FUNCTION_BLOCK "Station Selection"   // FB20, SCL
{ S7_Optimized_Access := 'TRUE' }
VERSION : 0.1
   VAR_IN_OUT
      settings : "Settings";
      stations : "Stations";
   END_VAR
   VAR
      firstStn : Int;
      rt : "Runtime Data";
      selectionExe : Bool;
      old : Struct
         prevGrp : Bool;
         nextGrp : Bool;
         stnSlct : Array[0..11] of Bool;
      END_STRUCT;
   END_VAR
   VAR_TEMP
      animate : USInt;
      btnPress : Bool;
      count : Int;
      currentBtn : Bool;
      evalObjCount : Int;
      i : Int;
      oldBtn : Bool;
      pStn : Int;
      stnName : WString;
      stnSelected : Bool;
      selState : Bool;
      selStnCount : Int;
      timerExpired : Bool;
      stnSelLblCount : Int;
   END_VAR
   VAR CONSTANT
      ptTimer : Real := 1.5;
   END_VAR
BEGIN
   REGION "UI INTERACTION ANIMATIONS"

       REGION "NEXT GROUP"
           #btnPress := #settings.stations.nextGroup.actuate;
           #animate := "Animate Bool"(colorTrue := "BgLGr",
                                      colorFalse := "BgGray",
                                      evalSignal := #btnPress);
           #settings.stations.nextGroup.animate := #animate;
       END_REGION

       REGION "PREVIOUS GROUP"
           #btnPress := #settings.stations.prevGroup.actuate;
           #animate := "Animate Bool"(colorTrue := "BgLGr",
                                      colorFalse := "BgGray",
                                      evalSignal := #btnPress);
           #settings.stations.prevGroup.animate := #animate;
       END_REGION

       REGION "SELECT ALL STATIONS"
           #btnPress := #settings.stations.selectAll.actuate;
           #animate := "Animate Bool"(colorTrue := "BgLGr",
                                      colorFalse := "BgGray",
                                      evalSignal := #settings.stations.selectAll.actuate);
           #settings.stations.selectAll.animate := #animate;
       END_REGION

   END_REGION

   REGION "POPULATE STATION LABELS"

       REGION "PROCESS NEXT GROUP PRESS"

           REGION "COPY TO LOCAL"
               #currentBtn := #settings.stations.nextGroup.actuate;
               #oldBtn := #old.nextGrp;
           END_REGION

           REGION "FALLING EDGE OF NEXT GROUP"
               IF NOT #currentBtn AND #oldBtn THEN

                   REGION "INCREMENT FIRST STATION"
                       #firstStn := #firstStn + 2;
                   END_REGION

                   REGION "UPPER LIMIT ROLL OVER"
                       IF #firstStn > "stnCount" THEN
                           #firstStn := #firstStn - "stnCount" - 1;
                       END_IF;
                   END_REGION

               END_IF;
           END_REGION

           REGION "NEXT GROUP CHANGE DETECTION"
               #old.nextGrp := #currentBtn;
           END_REGION

       END_REGION

       REGION "PROCESS PREVIOUS GROUP PRESS"

           REGION "COPY TO LOCAL"
               #currentBtn := #settings.stations.prevGroup.actuate;
               #oldBtn := #old.prevGrp;
           END_REGION

           REGION "FALLING EDGE OF PREVIOUS GROUP"
               IF NOT #currentBtn AND #oldBtn THEN

                   REGION "DECREMENT FIRST STATION"
                       #firstStn := #firstStn - 2;
                   END_REGION

                   REGION "LOWER LIMIT ROLL OVER"
                       IF #firstStn < 0 THEN
                           #firstStn := #firstStn + "stnCount" + 1;
                       END_IF;
                   END_REGION

               END_IF;
           END_REGION

           REGION "PREVIOUS GROUP CHANGE DETECTION"
               #old.prevGrp := #currentBtn;
           END_REGION

       END_REGION

       REGION "WRITE LABEL"

           REGION "COPY TO LOCAL"
               #evalObjCount := "hmiSelStnCount";
           END_REGION

           REGION "FOR EACH STATION SELECTION BUTTON"
               FOR #i := 0 TO #evalObjCount DO

                   REGION "CALCULATE POINTER"
                       #pStn := #firstStn + #i;
                   END_REGION

                   REGION "UPPER LIMIT ROLL OVER"
                       IF #pStn > "stnCount" THEN
                           #pStn := #firstStn + #i - "stnCount" - 1;
                       END_IF;
                   END_REGION

                   REGION "BUILD NAME"
                       #stnName := CONCAT_WSTRING(IN1 := #stations.me[#pStn].line,
                                                  IN2 := wstring#' ',
                                                  IN3 := "Strip Sign"(USINT_TO_WSTRING(#stations.me[#pStn].dropZone)));
                   END_REGION

                   REGION "WRITE NAME"
                       #settings.stations.selectBtns[#i].label := #stnName;
                   END_REGION

               END_FOR;
           END_REGION

       END_REGION

   END_REGION

   REGION "SINGLE STATION SELECTION"

       REGION "COPY TO LOCAL"
           #stnSelLblCount := "hmiSelStnCount";
       END_REGION

       REGION "LOOP THROUGH DISPLAYED STATIONS"
           FOR #i := 0 TO #stnSelLblCount DO

               REGION "CALCULATE POINTER"
                   #pStn := #firstStn + #i;
               END_REGION

               REGION "UPPER LIMIT ROLL OVER"
                   IF #pStn > "stnCount" THEN
                       #pStn := #firstStn + #i - "stnCount" - 1;
                   END_IF;
               END_REGION

               REGION "COPY TO LOCAL"
                   #currentBtn := #settings.stations.selectBtns[#i].actuate;
                   #oldBtn := #old.stnSlct[#i];
               END_REGION

               REGION "TOGGLE STATE ON FALLING EDGE"
                   IF NOT #currentBtn AND #oldBtn THEN
                       #selState := #stations.me[#pStn].settings.selected;
                       #selState := NOT #selState;
                       #stations.me[#pStn].settings.selected := #selState;
                   END_IF;
               END_REGION

               REGION "STATION SELECTION CHANGE DETECTION"
                   #old.stnSlct[#i] := #currentBtn;
               END_REGION

           END_FOR;
       END_REGION

   END_REGION

   REGION "MULTI SELECT TIMER"

       REGION "RUNTIME CALL"
           #rt.elapsed := RUNTIME(#rt.mem);
       END_REGION

       REGION "TIMER"

           REGION "COPY TO LOCAL"
               #btnPress := #settings.stations.selectAll.actuate;
           END_REGION

           REGION "ACCUMULATE RT VALUES"
               IF #btnPress THEN
                   #rt.asReal += LREAL_TO_REAL(#rt.elapsed);
               END_IF;
           END_REGION

           REGION "SET TIMER FLAG"
               IF #rt.asReal < #ptTimer THEN
                   #timerExpired := FALSE;
               END_IF;
               IF #rt.asReal >= #ptTimer THEN
                   #timerExpired := TRUE;
                   #rt.asReal := 0.0;
               END_IF;
           END_REGION

           REGION "RESET ACCUMULATED VALUE"
               IF NOT #btnPress THEN
                   #rt.asReal := 0.0;
                   #selectionExe := FALSE;
               END_IF;
           END_REGION

       END_REGION

   END_REGION

   REGION "EVALUATE MULTI SELECTION"
       IF #timerExpired AND NOT #selectionExe THEN

           REGION "COPY TO LOCAL"
               #selStnCount := #settings.stations.selCount;
           END_REGION

           REGION "SELECT ALL"
               IF #selStnCount < "stnCount" THEN
                   "Select Stations"(mode := TRUE,
                                     stations := #stations);
               END_IF;
           END_REGION

           REGION "DESELECT ALL"
               IF #selStnCount = "stnCount" THEN
                   "Select Stations"(mode := FALSE,
                                     stations := #stations);
               END_IF;
           END_REGION

           REGION "FLAG SELECTION EXECUTED"
               #selectionExe := TRUE;
           END_REGION

       END_IF;
   END_REGION

   REGION "SELECTION ANIMATIONS"

       REGION "COPY TO LOCAL"
           #stnSelLblCount := "hmiSelStnCount";
       END_REGION

       REGION "LOOP THROUGH BUTTONS"
           FOR #i := 0 TO #stnSelLblCount DO

               REGION "CALCULATE POINTER"
                   #pStn := #firstStn + #i;
               END_REGION

               REGION "UPPER LIMIT ROLL OVER"
                   IF #pStn > "stnCount" THEN
                       #pStn := #firstStn + #i - "stnCount" - 1;
                   END_IF;
               END_REGION

               REGION "COPY TO LOCAL"
                   #currentBtn := #settings.stations.selectBtns[#i].actuate;
                   #stnSelected := #stations.me[#pStn].settings.selected;
               END_REGION

               REGION "DRAW SELCTION HIGHLIGHTS"
                   #animate := "Animate Bool"(colorTrue := "BgLTe",
                                              colorFalse := "BgGray",
                                              evalSignal := #stnSelected);
               END_REGION

               REGION "ANIMATE BUTTON PRESS"
                   #animate := "Animate Bool"(colorTrue := "BgDTe",
                                              colorFalse := #animate,
                                              evalSignal := #currentBtn);
                   #settings.stations.selectBtns[#i].animate := #animate;
               END_REGION

           END_FOR;
       END_REGION

   END_REGION

   REGION "COUNT SELECTED STATIONS"

       REGION "INITIALIZE LOCAL"
           #count := 0;
           #evalObjCount := "stnCount";
       END_REGION

       REGION "LOOP THROUGH STATIONS"
           FOR #i := 0 TO #evalObjCount DO

               REGION "INCREMENT COUNT ON SELECTION"
                   #stnSelected := #stations.me[#i].settings.selected;
                   IF #stnSelected THEN
                       #count += 1;
                   END_IF;
               END_REGION

           END_FOR;
       END_REGION

       REGION "SAVE COUNT"
           #settings.stations.selCount := #count;
       END_REGION

   END_REGION
END_FUNCTION_BLOCK

FUNCTION_BLOCK "KP8 Button Selections"   // FB21, SCL
{ S7_Optimized_Access := 'TRUE' }
VERSION : 0.1
   VAR_INPUT
      reset : Bool;
   END_VAR
   VAR_IN_OUT
      settings : "Settings";
      stations : "Stations";
   END_VAR
   VAR
      enableState : Bool;
      oldBtnPresses : Array[0..7] of Bool;
      oldSelState : Array[0..7] of Bool;
      oldSelStnCount : Int;
      rt : "Runtime Data";
      timerExpired : Bool;
      selectionExe : Bool;
   END_VAR
   VAR_TEMP
      animate : USInt;
      btnPress : Bool;
      count : Int;
      i : Int;
      j : Int;
      mode : Bool;
      oldPress : Bool;
      pBtn : Int;
      selBtnCount : Int;
      selStnCount : Int;
      stnSelected : Bool;
   END_VAR
   VAR CONSTANT
      selectAllTime : Real := 1.5;
   END_VAR
BEGIN
   REGION "ENABLE KP8 BUTTON ASSIGNMENT SECTION"

       REGION "ENABLE"

           REGION "COPY TO LOCAL"
               #selStnCount := #settings.stations.selCount;
           END_REGION

           REGION "ON CHANGE IN SELECTED STATION COUNT"
               IF #selStnCount <> 0 AND #selStnCount <> #oldSelStnCount THEN

                   REGION "ENABLE KP8 SELECTIONS"
                       #enableState := TRUE;
                   END_REGION

               END_IF;
           END_REGION

       END_REGION

       REGION "DISABLE"

           REGION "COPY TO LOCAL"
               #selStnCount := #settings.stations.selCount;
           END_REGION

           REGION "ON DESELETION OF LAST STATION"
               IF #selStnCount = 0 AND #selStnCount <> #oldSelStnCount THEN

                   REGION "RESET ENABLED STATE"
                       #enableState := FALSE;
                   END_REGION

                   REGION "RESET BUTTON SELECTION STATES"
                       FOR #i := 0 TO "ptsPerStn" DO
                           #settings.kp8.btnSelState[#i] := FALSE;
                       END_FOR;
                   END_REGION

               END_IF;
           END_REGION

       END_REGION

   END_REGION

   REGION "SINGLE BUTTON SELECTION"

       REGION "LOOP THROUGH BUTTONS"
           FOR #i := 0 TO "ptsPerStn" DO

               REGION "EXCLUDE STOP RUNTIME AND RESET SELECTED BUTTONS"
                   IF #i <> 0 AND #i <> 4 THEN

                       REGION "COPY TO LOCAL"

                           REGION "CALCULATE BUTTON POINTER"
                               CASE #i OF
                                   1:
                                       #pBtn := 5;
                                   2:
                                       #pBtn := 3;
                                   3:
                                       #pBtn := 1;
                                   5:
                                       #pBtn := 4;
                                   6:
                                       #pBtn := 2;
                                   7:
                                       #pBtn := 0;
                                   ELSE
                                       ;
                               END_CASE;
                           END_REGION

                           #btnPress := #settings.kp8.buttons[#i].actuate OR #settings.viewingStation.btns[#pBtn].select.actuate;
                           #oldPress := #oldBtnPresses[#i];

                       END_REGION

                       REGION "TOGGLE STATE ON FALLING EDGE"
                           IF NOT #btnPress AND #oldPress THEN
                               #settings.kp8.btnSelState[#i] := NOT #settings.kp8.btnSelState[#i];
                               #settings.kp8.selBtnNumber := #i;
                           END_IF;
                       END_REGION

                       REGION "SAVE SELECTED BUTTON NUMBER ON DESELECT"
                           IF NOT #settings.kp8.btnSelState[#i] AND #oldSelState[#i] THEN
                               FOR #j := 0 TO "ptsPerStn" DO
                                   IF #settings.kp8.btnSelState[#j] THEN
                                       #settings.kp8.selBtnNumber := #j;
                                   END_IF;
                               END_FOR;
                           END_IF;
                       END_REGION

                       REGION "KP8 BUTON SELECTION CHANGE DETECTION"
                           #oldBtnPresses[#i] := #btnPress;
                       END_REGION

                   END_IF;
               END_REGION

           END_FOR;
       END_REGION

   END_REGION

   REGION "MULTI BUTTON SELECTION"

       REGION "MULTI SELECT TIMER"

           REGION "RUNTIME CALL"
               #rt.elapsed := RUNTIME(#rt.mem);
           END_REGION

           REGION "TIMER"

               REGION "COPY TO LOCAL"
                   #btnPress := #settings.kp8.selectButtons.actuate;
               END_REGION

               REGION "ACCUMULATE RT VALUES"
                   IF #btnPress THEN
                       #rt.asReal += LREAL_TO_REAL(#rt.elapsed);
                   END_IF;
               END_REGION

               REGION "SET TIMER FLAG"
                   IF #rt.asReal < #selectAllTime THEN
                       #timerExpired := FALSE;
                   END_IF;
                   IF #rt.asReal >= #selectAllTime THEN
                       #timerExpired := TRUE;
                       #rt.asReal := 0.0;
                   END_IF;
               END_REGION

               REGION "RESET ACCUMULATED VALUE"
                   IF NOT #btnPress THEN
                       #rt.asReal := 0.0;
                       #selectionExe := FALSE;
                   END_IF;
               END_REGION

           END_REGION

       END_REGION

       REGION "EVALUATE MULTI SELECTION"
           IF #timerExpired AND NOT #selectionExe THEN

               REGION "COPY TO LOCAL"
                   #selBtnCount := #settings.kp8.selCount;
               END_REGION

               REGION "SELECT ALL"
                   IF #selBtnCount < "ptsPerStn" - 1 THEN
                       #mode := TRUE;
                   END_IF;
               END_REGION

               REGION "DESELECT ALL"
                   IF #selBtnCount = "ptsPerStn" - 1 THEN
                       #mode := FALSE;
                   END_IF;
               END_REGION

               REGION "SAVE SELECTIONS"
                   FOR #i := 0 TO "ptsPerStn" DO

                       REGION "EXCLUDE STOP RUNTIME AND RESET SELECTED BUTTONS"
                           IF #i <> 0 AND #i <> 4 THEN

                               REGION "PERFROM SELECTION"
                                   #settings.kp8.btnSelState[#i] := #mode;
                               END_REGION

                           END_IF;
                       END_REGION

                   END_FOR;
               END_REGION

               REGION "SET SELECED BUTTON NUMBER TO 1"
                   #settings.kp8.selBtnNumber := 0;
               END_REGION

               REGION "FLAG SELECTION EXECUTED"
                   #selectionExe := TRUE;
               END_REGION

           END_IF;
       END_REGION
   END_REGION

   REGION "SAVE BUTTON SELECTIONS TO STATIONS"

       REGION "COPY TO LOCAL"
           #selStnCount := #settings.stations.selCount;
       END_REGION

       REGION "ON CHANGE IN BUTTON OR STATION SELECTON"
           IF #settings.kp8.btnSelState <> #oldSelState OR #selStnCount <> #oldSelStnCount THEN

               REGION "FOR SELECTED STATIONS"
                   FOR #i := 0 TO "stnCount" DO
                       #stnSelected := #stations.me[#i].settings.selected;
                       IF #stnSelected THEN

                           REGION "SAVE BUTTON SELECTION STATE"
                               #stations.me[#i].settings.btnSelection := #settings.kp8.btnSelState;
                           END_REGION

                       END_IF;
                   END_FOR;
               END_REGION

           END_IF;
       END_REGION

       REGION "SELECTED STATION COUNT CHANGE DETECTION"
           #oldSelStnCount := #selStnCount; 
       END_REGION

   END_REGION

   REGION "COUNT SELECTED BUTTONS"

       REGION "ON CHANGE IN BUTTON SELECTION STATES"
           IF #settings.kp8.btnSelState <> #oldSelState THEN

               REGION "INITIALIZE LOCAL"
                   #count := 0;
               END_REGION

               REGION "FOR EACH SELECTED BUTTON"
                   FOR #i := 0 TO "ptsPerStn" DO
                       IF #settings.kp8.btnSelState[#i] THEN

                           REGION "INCREMENT COUNT"
                               #count := #count + 1;
                           END_REGION

                       END_IF;
                   END_FOR;
               END_REGION

               REGION "SAVE COUNT"
                   #settings.kp8.selCount := #count;
               END_REGION

           END_IF;
       END_REGION

   END_REGION 

   REGION "UI INTERACTION ANIMATIONS"

       REGION "SELECT ALL BUTTONS"
           #btnPress := #settings.kp8.selectButtons.actuate;
           #animate := "Animate Bool"(colorTrue := "BgLGr",
                                      colorFalse := "BgGray",
                                      evalSignal := #btnPress);
           #settings.kp8.selectButtons.animate := #animate;
       END_REGION

       REGION "STOP RESET SELECTED STATION"
           #btnPress := #settings.kp8.buttons[0].actuate;
           #animate := "Animate Bool"(colorTrue := "FgGray",
                                      colorFalse := "BgGray",
                                      evalSignal := #btnPress);
           #settings.kp8.buttons[0].animate := #animate;
       END_REGION

       REGION "STOP RUNTIME"
           #btnPress := #settings.kp8.buttons[4].actuate;
           #animate := "Animate Bool"(colorTrue := "FgGray",
                                      colorFalse := "BgGray",
                                      evalSignal := #btnPress);
           #settings.kp8.buttons[4].animate := #animate;
       END_REGION

       REGION "BUTTON SELECTIONS"

           REGION "FOR EACH BUTTON"     
               FOR #i := 0 TO "ptsPerStn" DO

                   REGION "EXCLUDE STOP RUNTIME AND RESET SELECTED BUTTONS"
                       IF #i <> 0 AND #i <> 4 THEN

                           REGION "ANIMATE"

                               REGION "COPY TO LOCAL"
                                   #btnPress := #settings.kp8.buttons[#i].actuate;
                               END_REGION

                               REGION "ENABLE/DISABLE"
                                   #animate := "Animate Bool"(colorTrue := "BgGray",
                                                              colorFalse := "disabled",
                                                              evalSignal := #enableState);
                               END_REGION

                               REGION "ENABLED SUB ANIMATIONS"
                                   IF #enableState THEN

                                       REGION "BUTTON SELECTED"
                                           #animate := "Animate Bool"(colorTrue := "BgLTe",
                                                                      colorFalse := #animate,
                                                                      evalSignal := #settings.kp8.btnSelState[#i]);
                                       END_REGION

                                       REGION "BUTTON UP/DOWN"
                                           #animate := "Animate Bool"(colorTrue := "BgDTe",
                                                                      colorFalse := #animate,
                                                                      evalSignal := #btnPress);
                                       END_REGION
                                   END_IF;
                               END_REGION

                               REGION "SAVE ANIMATION"
                                   #settings.kp8.buttons[#i].animate := #animate;
                               END_REGION

                           END_REGION

                       END_IF;
                   END_REGION

               END_FOR;
           END_REGION

       END_REGION

   END_REGION

   REGION "DRAW KP8 BUTTON LABELS"
       IF #reset THEN
           #settings.kp8.buttons[1].label := wstring#'6';
           #settings.kp8.buttons[2].label := wstring#'4';
           #settings.kp8.buttons[3].label := wstring#'2';
           #settings.kp8.buttons[5].label := wstring#'5';
           #settings.kp8.buttons[6].label := wstring#'3';
           #settings.kp8.buttons[7].label := wstring#'1';
       END_IF;
   END_REGION

   REGION "CHANGE DETECTION"
       #oldSelState := #settings.kp8.btnSelState;
   END_REGION
END_FUNCTION_BLOCK

FUNCTION_BLOCK "Buffer Log: Part Requests"   // FB22, SCL
{ S7_Optimized_Access := 'TRUE' }
VERSION : 0.1
   VAR_INPUT
      stations : "Stations";
   END_VAR
   VAR_IN_OUT
      logBuffer : "Part Req Log";
      logFlag : Int;
   END_VAR
   VAR
      clpsLogTime : Real;
      old : Struct
         ordered : "Station Old Presses";
         requested : "Station Old Presses";
      END_STRUCT;
      pLogBuffer : Int;
      rt : "Runtime Data";
   END_VAR
   VAR_TEMP
      address : Int;
      btnCount : Int;
      clpsFlag : Bool;
      i : Int;
      j : Int;
      oldPartOrdered : Bool;
      oldPartReq : Bool;
      partOrdered : Bool;
      partReq : Bool;
      stnCount : Int;
      readTimeRetVal : Int;
      blankRow : "Part Req Log Row";
   END_VAR
   VAR CONSTANT
      clpsItrvl : Real := 2.0;
      fulfilled : Int := 3;
      ordered : Int := 2;
      requested : Int := 1;
   END_VAR
BEGIN
   REGION "RUNTIME CALL"
       #rt.elapsed := RUNTIME(#rt.mem);
       #rt.asReal := LREAL_TO_REAL(#rt.elapsed);
   END_REGION

   REGION "COPY TO LOCAL"
       #btnCount := "ptsPerStn";
       #stnCount := "stnCount";
   END_REGION

   REGION "FOR EACH STATION"
       FOR #i := 0 TO #stnCount DO

           REGION "FOR EACH BUTTON"
               FOR #j := 0 TO #btnCount DO

                   REGION "COPY TO LOCAL"
                       #partOrdered := #stations.me[#i].partOrdered[#j];
                       #partReq := #stations.me[#i].partRequested[#j];
                       #oldPartOrdered := #old.ordered.me[#i,#j];
                       #oldPartReq := #old.requested.me[#i,#j];
                   END_REGION;

                   REGION "CALCULATE ADDRESS"
                       #address := (#i + 1) * 10 + #j + 1;
                   END_REGION

                   REGION "ON PART REQUEST RISING EDGE"
                       IF #partReq AND NOT #oldPartReq THEN

                           REGION "LOG ENTRY"
                               #logBuffer.me[#pLogBuffer] := "Buffer Part Req Log Row: Generate"(address := #address,
                                                                                        type := #requested);
                           END_REGION

                           REGION "INCREMENT POINTER"
                               #pLogBuffer += 1;
                           END_REGION

                       END_IF;
                   END_REGION

                   REGION "ON PART ORDERED RISING EDGE"
                       IF #partOrdered AND NOT #oldPartOrdered THEN

                           REGION "REQUEST TYPE"
                               #logBuffer.me[#pLogBuffer] := "Buffer Part Req Log Row: Generate"(address := #address,
                                                                                                 type := #ordered);
                           END_REGION

                           REGION "INCREMENT POINTER"
                               #pLogBuffer += 1;
                           END_REGION

                       END_IF;
                   END_REGION

                   REGION "ON PART REQUEST FALLING EDGE"
                       IF NOT #partReq AND #oldPartReq THEN

                           REGION "REQUEST TYPE"
                               #logBuffer.me[#pLogBuffer] := "Buffer Part Req Log Row: Generate"(
                                   address := #address,
                                   type := #fulfilled
                               );
                           END_REGION

                           REGION "INCREMENT POINTER"
                               #pLogBuffer += 1;
                           END_REGION

                       END_IF;
                   END_REGION

                   REGION "SAVE FOR CHANGE DETECTION"
                       #old.requested.me[#i, #j] := #partReq;
                       #old.ordered.me[#i, #j] := #partOrdered;
                   END_REGION

               END_FOR;
           END_REGION

       END_FOR;
   END_REGION

   REGION "SEND TO HMI"

       REGION "ON ENTRY IN BUFFER"
           IF #logBuffer.me[0].address <> 0 THEN

               REGION "TIMER"
                   #clpsLogTime += #rt.asReal;
                   IF #clpsLogTime >= #clpsItrvl THEN
                       #clpsLogTime := 0.0;
                       #clpsFlag := TRUE;
                   END_IF;
               END_REGION

               REGION "EXECUTE COLLAPSE"
                   IF #clpsFlag THEN

                       REGION "MOVE BUFFER UP ONE POSITION"
                           FOR #i := 0 TO 98 DO
                               #logBuffer.me[#i] := #logBuffer.me[#i + 1];
                           END_FOR;
                       END_REGION

                       REGION "DELETE LAST ROW"
                           #logBuffer.me[99] := #blankRow;
                       END_REGION

                       REGION "FLAG FOR HMI"
                           #logFlag += 1;
                           IF #logFlag > 9 THEN
                               #logFlag := 0;
                           END_IF;
                       END_REGION

                       REGION "DECREMENT POINTER"
                           #pLogBuffer -= 1;
                       END_REGION

                   END_IF;
               END_REGION

           END_IF;
       END_REGION

   END_REGION

   REGION "RESET TIMER"
       IF #logBuffer.me[0].address = 0 THEN
           #clpsLogTime := 0.0;
       END_IF;
   END_REGION
END_FUNCTION_BLOCK

FUNCTION_BLOCK "Enable Assignment Pair"   // FB23, SCL
{ S7_Optimized_Access := 'TRUE' }
VERSION : 0.1
   VAR_INPUT
      disable : Bool;
      enable : Bool;
   END_VAR
   VAR_IN_OUT
      value : WString;
      assignAnimate : USInt;
      ioFieldAnimate : USInt;
   END_VAR
   VAR
      old : Struct
         disabled : Bool;
         enabled : Bool;
      END_STRUCT;
   END_VAR
BEGIN
   REGION "DISABLED"    
       IF #disable THEN
           #value := wstring#'';
           #assignAnimate := "disabled";
           #ioFieldAnimate := "disabled";
       END_IF;
   END_REGION

   REGION "ENABLED"
           IF #enable THEN
               #assignAnimate := "BgGray";
               #ioFieldAnimate := "BgWh";
           END_IF;
   END_REGION
END_FUNCTION_BLOCK

FUNCTION_BLOCK "Assign Button Parameters"   // FB24, SCL
{ S7_Optimized_Access := 'TRUE' }
VERSION : 0.1
   VAR_INPUT
      settings : "Settings";
   END_VAR
   VAR_IN_OUT
      stations : "Stations";
   END_VAR
   VAR
      old : Struct
         allotted : Bool;
         critical : Bool;
         pn : Bool;
      END_STRUCT;
   END_VAR
   VAR_TEMP
      assign : Bool;
      btn : Struct
         allotted : Bool;
         critical : Bool;
         pn : Bool;
      END_STRUCT;
      btnSelected : Bool;
      i : Int;
      j : Int;
      partNumber : WString;
      stnSelected : Bool;
      timerReal : Real;
   END_VAR
BEGIN
   REGION "COPY TO LOCACL"
       #btn.allotted := #settings.alotted.assign.actuate;
       #btn.critical := #settings.critical.assign.actuate;
       #btn.pn := #settings.partNumber.assign.actuate;
   END_REGION

   REGION "ASSIGNMENT PULSE"
       #assign := (#btn.allotted AND NOT #old.allotted)
                   OR (#btn.critical AND NOT #old.critical)
                   OR (#btn.pn AND NOT #old.pn);
   END_REGION

   REGION "ON ASSIGNMENT PULSE"
       IF #assign THEN
           REGION "PROCESS VARIABLE"

               REGION "PART NUMBER"
                   IF #btn.pn THEN
                       #partNumber := #settings.partNumber.ioField.value;
                   END_IF;
               END_REGION

               REGION "CRITICAL TIME"
                   IF #btn.critical THEN
                       #timerReal := "WString Timer to Real"(#settings.critical.ioField.value);
                   END_IF;
               END_REGION

               REGION "ALLOTTED TIME"
                   IF #btn.allotted THEN
                       #timerReal := "WString Timer to Real"(#settings.alotted.ioField.value);
                   END_IF;
               END_REGION

           END_REGION

           REGION "FOR EACH STATION"
               FOR #i := 0 TO "stnCount" DO

                   REGION "COPY TO LOCAL"
                       #stnSelected := #stations.me[#i].settings.selected;
                   END_REGION

                   REGION "ON SELECTED STATION"
                       IF #stnSelected THEN

                           REGION "FOR EACH BUTTON"
                               FOR #j := 0 TO "ptsPerStn" DO

                                   REGION "COPY TO LOCAL"
                                       #btnSelected := #stations.me[#i].settings.btnSelection[#j];
                                   END_REGION

                                   REGION "ON SELECTED BUTTON"
                                       IF #btnSelected THEN

                                           REGION "ASSIGN PART NUMBER"
                                               IF #btn.pn THEN
                                                   #stations.me[#i].partNumbers[#j] := #partNumber;
                                               END_IF;
                                           END_REGION

                                           REGION "ASSIGN ALLOTTED TIME"
                                               IF #btn.allotted THEN
                                                   #stations.me[#i].presetTime.allotted[#j] := #timerReal;
                                               END_IF;
                                           END_REGION

                                           REGION "ASSIGN CRITICAL TIME"
                                               IF #btn.critical THEN
                                                   #stations.me[#i].presetTime.critical[#j] := #timerReal;
                                               END_IF;
                                           END_REGION

                                       END_IF;
                                   END_REGION

                               END_FOR;
                           END_REGION

                       END_IF;
                   END_REGION

               END_FOR;
           END_REGION

       END_IF;
   END_REGION

   REGION "CHANGE DETECTION"
       #old := #btn;
   END_REGION
END_FUNCTION_BLOCK

FUNCTION_BLOCK "Animate: PN & Timers"   // FB25, SCL
{ S7_Optimized_Access := 'TRUE' }
VERSION : 0.1
   VAR_INPUT
      stations : "Stations";
   END_VAR
   VAR_IN_OUT
      settings : "Settings";
   END_VAR
   VAR
      instPNEntEnable : "Enable Assignment Pair";
      instAlltEntEnable : "Enable Assignment Pair";
      instCrtEntEnable : "Enable Assignment Pair";
   END_VAR
   VAR_TEMP
      animate : USInt;
      disable : Bool;
      enable : Bool;
      selBtnCount : Int;
      selStnCount : Int;
   END_VAR
BEGIN
   REGION "COPY TO LOCAL"
       #selBtnCount := #settings.kp8.selCount;
       #selStnCount := #settings.stations.selCount;
   END_REGION

   REGION "ENABLE/DISABLE FOR PN AND TIMERS"

       REGION "SET DISABLE"
           IF #selStnCount = 0 OR #selBtnCount = 0 THEN
               #disable := TRUE;
               #enable := FALSE;
           END_IF;
       END_REGION

       REGION "SET ENABLE"
           IF #selStnCount <> 0 AND #selBtnCount <> 0 THEN
               #disable := FALSE;
               #enable := TRUE;
           END_IF;
       END_REGION

   END_REGION

   REGION "PN ANIMATION FUNCTIONS"
       #animate := #settings.partNumber.assign.animate;
       #instPNEntEnable(disable := #disable,
                        enable := #enable,
                        value := #settings.partNumber.ioField.value,
                        assignAnimate := #animate,
                        ioFieldAnimate := #settings.partNumber.ioField.animate);
       #animate := "Animate Bool"(colorTrue := "BgLGr",
                                  colorFalse := #animate,
                                  evalSignal := #settings.partNumber.assign.actuate);
       #settings.partNumber.assign.animate := #animate;
   END_REGION

   REGION "ALLOTTED TIME ANIMATION FUNCTIONS"
       #animate := #settings.alotted.assign.animate;
       #instAlltEntEnable(disable := #disable,
                          enable := #enable,
                          value := #settings.alotted.ioField.value,
                          assignAnimate := #animate,
                          ioFieldAnimate := #settings.alotted.ioField.animate);
       #animate := "Animate Bool"(colorTrue := "BgLGr",
                                  colorFalse := #animate,
                                  evalSignal := #settings.alotted.assign.actuate);
       #settings.alotted.assign.animate := #animate;
   END_REGION

   REGION "CRITICAL TIME ANIMATION FUNCTIONS"
       #animate := #settings.critical.assign.animate;
       #instCrtEntEnable(disable := #disable,
                         enable := #enable,
                         value := #settings.critical.ioField.value,
                         assignAnimate := #animate,
                         ioFieldAnimate := #settings.critical.ioField.animate);
       #animate := "Animate Bool"(colorTrue := "BgLGr",
                                  colorFalse := #animate,
                                  evalSignal := #settings.critical.assign.actuate);
       #settings.critical.assign.animate := #animate;
   END_REGION
END_FUNCTION_BLOCK

FUNCTION_BLOCK "Global to Sim"   // FB26, SCL
{ S7_Optimized_Access := 'TRUE' }
VERSION : 0.1
   VAR_INPUT
      stations : "Stations";
   END_VAR
   VAR_IN_OUT
      simStations : "Simulated Stations";
   END_VAR
   VAR
      old : Struct
         nextGrp : Bool;
         prevGrp : Bool;
      END_STRUCT;
   END_VAR
   VAR_TEMP
      animate : USInt;
      btnCount : Int;
      currentBtn : Bool;
      dzLabel : WString;
      firstStn : Int;
      i : Int;
      intBox : Int;
      j : Int;
      kp8Color : DWord;
      label : WString;
      oldBtn : Bool;
      pSim : Int;
      pStn : Int;
      simKP8Count : Int;
      stnCount : Int;
   END_VAR
   VAR CONSTANT
      space : WString := WSTRING#' ';
      lead0 : WString := WSTRING#'0';
      volvo16 : WString := WSTRING#'VOLVO 16';
   END_VAR
BEGIN
   REGION "COPY TO LOCAL"
       #btnCount := "ptsPerStn";
       #firstStn := #simStations.firstStn;
       #stnCount := "stnCount";
       #simKP8Count := "simKP8Count";
   END_REGION

   REGION "RESOLVE STATION POINTER"

       REGION "PROCESS NEXT GROUP PRESS"

           REGION "COPY TO LOCAL"
               #currentBtn := #simStations.down.actuate;
               #oldBtn := #old.nextGrp;
           END_REGION

           REGION "FALLING EDGE OF NEXT GROUP"
               IF NOT #currentBtn AND #oldBtn THEN

                   REGION "INCREMENT FIRST STATION"
                       #firstStn += #simKP8Count;
                   END_REGION

                   REGION "UPPER LIMIT ROLL OVER"
                       IF #firstStn > #stnCount THEN
                           #firstStn -= #stnCount + 1;
                       END_IF;
                   END_REGION

               END_IF;
           END_REGION

           REGION "NEXT GROUP CHANGE DETECTION"
               #old.nextGrp := #currentBtn;
           END_REGION

       END_REGION

       REGION "PROCESS PREVIOUS GROUP PRESS"

           REGION "COPY TO LOCAL"
               #currentBtn := #simStations.up.actuate;
               #oldBtn := #old.prevGrp;
           END_REGION

           REGION "FALLING EDGE OF PREVIOUS GROUP"
               IF NOT #currentBtn AND #oldBtn THEN

                   REGION "DECREMENT FIRST STATION"
                       #firstStn -= #simKP8Count;
                   END_REGION

                   REGION "LOWER LIMIT ROLL OVER"
                       IF #firstStn < 0 THEN
                           #firstStn += #stnCount + 1;
                       END_IF;
                   END_REGION

               END_IF;
           END_REGION

           REGION "PREVIOUS GROUP CHANGE DETECTION"
               #old.prevGrp := #currentBtn;
           END_REGION

       END_REGION

   END_REGION

   REGION "FOR EACH BUTTON"
       FOR #i := 0 TO 11 DO

           REGION "CALCULATE POINTER"
               #pStn := #i + #firstStn;
               #pSim := #i;
           END_REGION

           REGION "UPPER LIMIT ROLL OVER"
               IF #pStn > #stnCount THEN
                   #pStn := #firstStn + #i - #stnCount - 1;
               END_IF;
           END_REGION

           REGION "COPY TO LOCAL"
               #kp8Color := #stations.me[#pStn].kp8Out;
           END_REGION

           REGION "LABEL STATIONS"

               REGION "DETERMINE LINE LABEL"
                   #label := #stations.me[#pStn].line;
                   IF #label = #volvo16 THEN
                       #label := WSTRING#'V16';
                   END_IF;
               END_REGION

               REGION "DETERMINE DROP ZONE LABEL"
                   #intBox := USINT_TO_INT(#stations.me[#pStn].dropZone);
                   IF #intBox <= 9 THEN
                       #dzLabel := CONCAT_WSTRING(IN1 := #lead0,
                                                  IN2 := "Strip Sign"(INT_TO_WSTRING(#intBox)));
                   END_IF;
                   IF #intBox >= 10 THEN
                       #dzLabel := "Strip Sign"(INT_TO_WSTRING(#intBox));
                   END_IF;
               END_REGION

               REGION "WRITE LABEL"
                   #label := CONCAT_WSTRING(IN1 := #label,
                                            IN2 := #space,
                                            IN3 := #dzLabel);
                   #simStations.me[#pSim].stn.label := #label;
               END_REGION

           END_REGION

           REGION "ANIMATE STATION LABEL"
               #simStations.me[#pSim].stn.animate := "BgGray";
           END_REGION

           REGION "FOR EACH BUTTON"
               FOR #j := 0 TO #btnCount DO

                   REGION "COLOR BUTTONS"
                       #animate := "KP8 Color to Sim Animation"(kp8Color := #kp8Color,
                                                                btnNumber := #j);
                       #simStations.me[#pSim].btn.animate[#j] := #animate;
                   END_REGION

                   REGION "WRITE BUTTON LABELS"
                       #intBox := "Pointer Calc: KP8 Labels"(#j);
                       #label := "Strip Sign"(INT_TO_WSTRING(#intBox));
                       #simStations.me[#pSim].btn.labels[#j] := #label;
                   END_REGION

               END_FOR;
           END_REGION

       END_FOR;
   END_REGION

   REGION "SAVE FIRST STATION"
       #simStations.firstStn := #firstStn;
   END_REGION

   REGION "ANIMATE NEXT GROUP PRESS"
       #simStations.down.animate := "Animate Bool"(colorTrue := "BgLGr",
                                                   colorFalse := "BgGray",
                                                   evalSignal := #simStations.down.actuate);
   END_REGION

   REGION "ANIMATE PREV GROUP PARESS"
       #simStations.up.animate := "Animate Bool"(colorTrue := "BgLGr",
                                                 colorFalse := "BgGray",
                                                 evalSignal := #simStations.up.actuate);
   END_REGION
END_FUNCTION_BLOCK

FUNCTION_BLOCK "NetDiag: Get IPs"   // FB27, SCL
{ S7_Optimized_Access := 'TRUE' }
VERSION : 0.1
   VAR_OUTPUT
      error : Bool := FALSE;   // Rising edge informs that an error occurred during the execution of the FB
      status : Word := 16#0000;   // Current status of FB
      statusID : Word := 16#0;   // Current status ID of calling instruction
   END_VAR
   VAR_IN_OUT
      ioSystemData : "UserDiag_typeIOSystem";   // IO-System diagnostics data
   END_VAR
   VAR
      statError : Bool := FALSE;   // Static value for output error
      statStatus : Word := 16#0000;   // Static value for output status
      statStatusID : Word := 16#0;   // Static value for output statusID
      instGetStationInfo : GetStationInfo;   // Instance of GetStationInfo
      statFirstDeviceFlag : Bool := TRUE;   // Help tag for the first device in the linked list
      statDeviceIndex : Int := 0;   // Device/slave index
   END_VAR
   VAR_TEMP
      tempIP : IF_CONF_v4;   // Temporary IP address
   END_VAR
   VAR CONSTANT
      STATUS_EXECUTION_FINISHED : Word := 16#0000;   // Execution finished without errors
      ID_GET_STATION_INFO : Word := 12;   // StatusID during GetStationInfo command
      MODE_IPV4 : UInt := 1;   // Address parameter according to IPv4
      LAST_DEVICE : Int := -1;   // No next device
   END_VAR
BEGIN
   //=============================================================================
   //SIEMENS AG
   //(c)Copyright 2015 All Rights Reserved
   //-----------------------------------------------------------------------------
   //Library: 
   //Tested with: S7-1516-3 PN/DP FW 2.5
   //Engineering: TIA Portal V15
   //Restrictions: Call in cyclic OB
   //Requirements: -
   //Functionality: Get IP address of IO devices
   //-----------------------------------------------------------------------------
   //Change log table:
   //Version  Date       Expert in charge                Changes applied
   //01.00.00 20.12.2017 Siemens Industry Online Support First released version
   //=============================================================================

   //=============================================================================
   // Go through existing devices and get IP address
   //=============================================================================
   // Initialize the pointer for the first run 
   IF (#statFirstDeviceFlag = TRUE)
   THEN
       #statDeviceIndex := #ioSystemData.firstDevice;
       #statFirstDeviceFlag := FALSE;
   END_IF;

   // Check and store the IP address, if the device is existing
   // GetStationInfo is an acyclic instruction. In the FB, the
   // instruction has to be repeated until it is done or error
   IF ((#ioSystemData.number >= 100)
       AND (#ioSystemData.number <= 115)
       AND (#ioSystemData.devices[#statDeviceIndex].exists = TRUE)
       AND (#ioSystemData.devices[#statDeviceIndex].ipAddress.ADDR[1] = 0))
   THEN
       // Get IP address of each decive in PN System
       #instGetStationInfo(REQ := TRUE,
                           LADDR := #ioSystemData.devices[#statDeviceIndex].hardwareId,
                           MODE := #MODE_IPV4,
                           DATA := #tempIP);

       IF (#instGetStationInfo.ERROR = TRUE)
       THEN
           // Error handling
           #statStatus := #instGetStationInfo.STATUS;
           #statStatusID := #ID_GET_STATION_INFO;
           #statError := TRUE;

           // Everything is ok --> Copy IP address    
       ELSIF (#instGetStationInfo.DONE = TRUE)
       THEN
           #ioSystemData.devices[#statDeviceIndex].ipAddress := #tempIP.InterfaceAddress;

           // Initialize the pointer for the next run
           #statDeviceIndex := #ioSystemData.devices[#statDeviceIndex].nextDevice;
       ELSE
           ;
       END_IF;
   ELSE
       // Initialize the pointer for the next run
       #statDeviceIndex := #ioSystemData.devices[#statDeviceIndex].nextDevice;
   END_IF;

   // Check last device
   IF (#statDeviceIndex = #LAST_DEVICE)
   THEN
       #statDeviceIndex := #ioSystemData.firstDevice;
   END_IF;

   // Write static values to outputs
   #error := #statError;
   #status := #statStatus;
   #statusID := #statStatusID;
END_FUNCTION_BLOCK

FUNCTION_BLOCK "NetDiag: Coordinate"   // FB28, LAD
{ S7_Optimized_Access := 'TRUE' }
VERSION : 0.1
// //============================================================================
// //SIEMENS AG
// //(c)Copyright 2017 All Rights Reserved
// //-----------------------------------------------------------------------------
// //Library: -
// //Tested with: S7-1516-3 PN/DP FW 2.5
// //Engineering: TIA Portal V15
// //Restrictions: -
// //Requirements: -
// //Functionality: Main FB for diagnostics
// //-----------------------------------------------------------------------------
// //Change log table:
// //Version  Date              Expert in charge                               Changes applied
// //01.00.00 25.04.2017 Siemens Industry Online Support First released version
// //01.01.00 01.12.2017 Siemens Industry Online Support Renamed in "UserDiag_Diagnostics"
// //                                                                                                    Check Flag "startDiag"
// //============================================================================
   VAR_IN_OUT
      startDiag : Bool := false;   // Startflag for diagnostic
      plcData : "UserDiag_typePLC";   // PLC diagnostics data
      ioSystemData : Array[1.."USERDIAG_IO_SYSTEMS_UPPER_LIM"] of "UserDiag_typeIOSystem";   // IO-System diagnostics data
   END_VAR
   VAR
      instPLCChk : "NetDiag: Check PLC";   // Instance of "UserDiag_PLCCheck"
      instIOSysChk : "NetDiag: IO Systems";   // Instance of "UserDiag_IOSystemCheck"
   END_VAR
BEGIN

REGION Network 1: Check Startflag for diagnostic
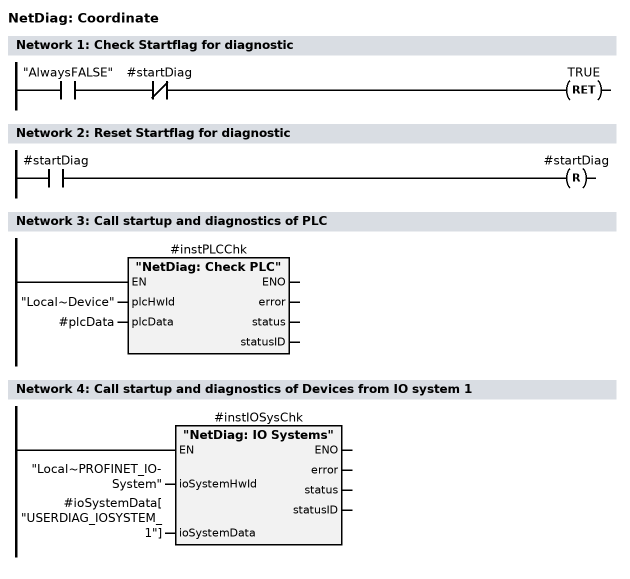
   IF "AlwaysFALSE" AND NOT #startDiag THEN
       ENO := TRUE;
       RETURN;
   END_IF;
END_REGION

REGION Network 2: Reset Startflag for diagnostic
   RUNG wire#powerrail
      Contact( #startDiag )
      R_Coil( #startDiag )
   END_RUNG
   // the same network as SCL:
   IF #startDiag THEN #startDiag := FALSE; END_IF;
END_REGION

REGION Network 3: Call startup and diagnostics of PLC
   RUNG wire#powerrail
      #instPLCChk(plcHwId := "Local~Device", plcData := #plcData, error =>, status =>, statusID =>)
   END_RUNG
   // the same network as SCL:
   #instPLCChk(plcHwId := "Local~Device", plcData := #plcData);   // "NetDiag: Check PLC"
END_REGION

REGION Network 4: Call startup and diagnostics of Devices from IO system 1
   RUNG wire#powerrail
      #instIOSysChk(ioSystemHwId := "Local~PROFINET_IO-System", ioSystemData := #ioSystemData["USERDIAG_IOSYSTEM_1"], error =>, status =>, statusID =>)
   END_RUNG
   // the same network as SCL:
   #instIOSysChk(ioSystemHwId := "Local~PROFINET_IO-System",   // "NetDiag: IO Systems"
                 ioSystemData := #ioSystemData["USERDIAG_IOSYSTEM_1"]);
END_REGION
END_FUNCTION_BLOCK

FUNCTION_BLOCK "NetDiag: Check PLC"   // FB29, SCL
{ S7_Optimized_Access := 'TRUE' }
VERSION : 0.1
   VAR_INPUT
      plcHwId : Hw_Device := 0;   // Hardware ID
   END_VAR
   VAR_OUTPUT
      error : Bool := FALSE;   // Rising edge informs that an error occurred during the execution of the FB
      status : Word := 16#0000;   // Current status of FB
      statusID : Word := 16#0;   // Current status ID of calling instruction
   END_VAR
   VAR_IN_OUT
      plcData : "UserDiag_typePLC";   // PLC diagnostics data
   END_VAR
   VAR
      statError : Bool := FALSE;   // Static value for output error
      statStatus : Word := 16#0000;   // Static value for output status
      statStatusID : Word := 16#0;   // Static value for output statusID
      statGeoAddr : GEOADDR;   // Slot information
      statGeoLaddr : Hw_Any := 16#0000;   // GEO2LOG hardware identifier
      statProblemPlcModulStates : Array[0..#MODULES_STATES_UPPER_LIM] of Bool;   // Storage of the status of all modules in the PLC central station --> State: Problem
      statFaultyPlcModulStates : Array[0..#MODULES_STATES_UPPER_LIM] of Bool;   // Storage of the status of all modules in the PLC central station --> State: Faulty
      statExistingPlcModulStates : Array[0..#MODULES_STATES_UPPER_LIM] of Bool;   // Storage of the status of all modules in the PLC central station --> State: Exists
      statActualCentralModules : USInt := 0;   // Actual number of modules in the central station (PLC)
   END_VAR
   VAR_TEMP
      tempSlotNum : Int;   // Index slot number
      tempRetValGeo : Int;   // GEO2LOG error information
      tempRetValModuleStates : Int;   // Return value system function ModuleStates
   END_VAR
   VAR CONSTANT
      STATUS_EXECUTION_FINISHED : Word := 16#0000;   // Execution finished without errors
      ERR_MAX_SLOTS_PER_PLC : Word := 16#8400;   // There are more modules configured as defined with the user constant: USERDIAG_SLOTS_PER_PLC_UPPER_LIM
      ID_LOCAL : Word := 1;   // StatusID local
      ID_MODULE_STATES_CONFIGURED : Word := 2;   // StatusID during ModuleStates command (configured mode)
      ID_MODULE_STATES_FAULTY : Word := 3;   // StatusID during ModuleStates command (faulty mode)
      ID_MODULE_STATES_PROBLEM : Word := 4;   // StatusID during ModuleStates command (problem mode)
      ID_MODULE_STATES_EXISTING : Word := 5;   // StatusID during ModuleStates command (existing mode)
      ID_LED : Word := 12;   // StatusID occurred during LED command
      MODE_FAULTY : USInt := 2;   // Used for instruction DeviceStates, read out all faulty devices
      MODE_EXIST : USInt := 4;   // Used for instruction DeviceStates, read out all devices not reachable
      MODE_PROBLEM : USInt := 5;   // Used for instruction DeviceStates, read out all devices with several problems
      STATE_OK : USInt := 1;   // Module state: ok
      STATE_FAULT : USInt := 2;   // Modulestate: fault
      STATE_PROBLEM : USInt := 5;   // Module state: problem
      STATE_WAS_FAULT : USInt := 12;   // Module state: was fault
      STATE_PROBLEM_GONE : USInt := 15;   // Module state: had a problem
      MODULE_OF_PLC : USInt := 4;   // GEO2LOG structure: HW type = 4
      CPU : USInt := 0;   // GEO2LOG structure: Area = 0
      CENTRAL_SYSTEM : USInt := 0;   // GEO2LOG structure: IO System = 0
      CENTRAL_STATION : USInt := 0;   // GEO2LOG structure: Station = 0
      NO_LED : Int := 0;   // LED does not exist
      LED_OFF : Int := 1;   // LED is permanently switched off
      LED_NO_INFO : Int := 9;   // LED exists, but status information not available
      MODULES_STATES_UPPER_LIM : Int := 127;   // Upper array limit for output tag of instruction ModuleStates
      ERROR_LED : UInt := 2;   // Identification number of the LED
   END_VAR
BEGIN
   //=============================================================================
   //SIEMENS AG
   //(c)Copyright 2017 All Rights Reserved
   //-----------------------------------------------------------------------------
   //Library: 
   //Tested with: S7-1516-3 PN/DP FW 2.5
   //Engineering: TIA Portal V15
   //Restrictions: Call in cyclic OB
   //Requirements: -
   //Functionality: Determine plc state and local module states
   //-----------------------------------------------------------------------------
   //Change log table:
   //Version  Date       Expert in charge                Changes applied
   //01.00.00 27.01.2017 Siemens Industry Online Support First released version
   //01.00.01 20.12.2017 Siemens Industry Online Support actualConfiguredSlots >= 1
   //01.00.02 27.02.2018 Siemens Industry Online Support Minor corrections
   //=============================================================================

   IF (#plcData.hardwareId = 0)
   THEN
       #statGeoAddr.HWTYPE := #MODULE_OF_PLC;      // Hardware type 4: module
       #statGeoAddr.AREA := #CPU;                  // Area ID 0: CPU
       #statGeoAddr.IOSYSTEM := #CENTRAL_SYSTEM;   // PROFINET IO system (0 = central unit in the rack)
       #statGeoAddr.STATION := #CENTRAL_STATION;   // Number of the rack if area identifier AREA = 0 (central module)

       #statStatus := #STATUS_EXECUTION_FINISHED;
       #statStatusID := 0;
       #statError := FALSE;
       #statActualCentralModules := 0;

       FOR #tempSlotNum := 0 TO "USERDIAG_SLOTS_PER_PLC_UPPER_LIM" DO
           // Slot number
           #statGeoAddr.SLOT := INT_TO_UINT(#tempSlotNum);
           // read LADDR from local modules
           #tempRetValGeo := GEO2LOG(GEOADDR := #statGeoAddr,
                                     LADDR => #statGeoLaddr);
           // Check Retval
           IF ((#tempRetValGeo = 0)
               AND (#statGeoLaddr <> 16#0))
           THEN
               // Store LADDR from local modules in diagnostic data block
               IF (#tempSlotNum = 1)
               THEN
                   #plcData.hardwareId := #statGeoLaddr;
               END_IF;
               #plcData.slots[#tempSlotNum].hardwareId := #statGeoLaddr;
               #statActualCentralModules := #statActualCentralModules + 1;
               #plcData.slots[#tempSlotNum].configured := TRUE;
           ELSE
               // If the return value ist not = 0 --> the device/system/module is not
               // configured --> No error handling
               // set LADDR from local modules to 0 in diagnostic data block
               #plcData.slots[#tempSlotNum].hardwareId := 0;
               #plcData.slots[#tempSlotNum].configured := FALSE;
           END_IF;
           // Store the actual configured devices in the diagnostics DB
           #plcData.actualConfiguredSlots := #statActualCentralModules;
       END_FOR;

       // Check if further slots are configured
       #statGeoAddr.SLOT := INT_TO_UINT(#tempSlotNum);

       #tempRetValGeo := GEO2LOG(GEOADDR := #statGeoAddr,
                                 LADDR => #statGeoLaddr);

       IF ((#tempRetValGeo = 0)
           AND (#statGeoLaddr <> 16#0))
       THEN
           // In the PLC are more slots configured as defined with the user constant
           #statStatus := #ERR_MAX_SLOTS_PER_PLC;
           #statStatusID := #ID_LOCAL;
           #statError := TRUE;
       END_IF;

   END_IF;

   // Reset PLC error state
   #plcData.error := FALSE;

   //=============================================================================
   // Check modul states from LOCAL MODULES
   //=============================================================================
   // Check if central module are available - at least one module is always
   // configured, the PLC itself
   IF (#plcData.actualConfiguredSlots >= 1)
   THEN

       // Check the status of the local modules
       #tempRetValModuleStates := ModuleStates(LADDR := #plcHwId,
                                               MODE := #MODE_PROBLEM,
                                               STATE := #statProblemPlcModulStates);

       // Check if the block call was successful
       IF (#tempRetValModuleStates <> 0)
       THEN
           // Error handling
           #statStatus := INT_TO_WORD(#tempRetValModuleStates);
           #statStatusID := #ID_MODULE_STATES_PROBLEM;
           #statError := TRUE;
       ELSE
           ; // Everything is ok!
       END_IF;

       #tempRetValModuleStates := ModuleStates(LADDR := #plcHwId,
                                               MODE := #MODE_FAULTY,
                                               STATE := #statFaultyPlcModulStates);

       // Check if the block call was successful
       IF (#tempRetValModuleStates <> 0)
       THEN
           // Error handling
           #statStatus := INT_TO_WORD(#tempRetValModuleStates);
           #statStatusID := #ID_MODULE_STATES_FAULTY;
           #statError := TRUE;
       ELSE
           ; // Everything is ok!
       END_IF;

       #tempRetValModuleStates := ModuleStates(LADDR := #plcHwId,
                                               MODE := #MODE_EXIST,
                                               STATE := #statExistingPlcModulStates);

       // Check if the block call was successful
       IF (#tempRetValModuleStates <> 0)
       THEN
           // Error handling
           #statStatus := INT_TO_WORD(#tempRetValModuleStates);
           #statStatusID := #ID_MODULE_STATES_EXISTING;
           #statError := TRUE;
       ELSE
           ; // Everything is ok!
       END_IF;

   ELSE
       ; // There are no central moduls configured
   END_IF;

   //=============================================================================
   // Set module states of LOCAL MODULES
   //=============================================================================
   #tempSlotNum := 0;
   WHILE (#tempSlotNum <= #plcData.actualConfiguredSlots)
   DO
       IF (#plcData.slots[#tempSlotNum].configured)
       THEN
           IF (#statExistingPlcModulStates[#tempSlotNum + 1] = TRUE)
           THEN
               #plcData.slots[#tempSlotNum].exists := TRUE;
               CASE #plcData.slots[#tempSlotNum].state OF
                   #STATE_WAS_FAULT,
                   #STATE_PROBLEM_GONE:
                       ;
                   #STATE_FAULT:
                       #plcData.slots[#tempSlotNum].state := #STATE_WAS_FAULT;
                   #STATE_PROBLEM:
                       #plcData.slots[#tempSlotNum].state := #STATE_PROBLEM_GONE;
                   ELSE
                       #plcData.slots[#tempSlotNum].state := #STATE_OK;
               END_CASE;
           ELSE
               #plcData.slots[#tempSlotNum].error := TRUE;
               #plcData.error := TRUE;
               #plcData.slots[#tempSlotNum].exists := FALSE;
           END_IF;

           IF (#statFaultyPlcModulStates[#tempSlotNum + 1] = TRUE)
           THEN
               // Modul is faulty
               #plcData.slots[#tempSlotNum].faulty := TRUE;
               #plcData.slots[#tempSlotNum].problem := TRUE;
               #plcData.slots[#tempSlotNum].error := TRUE;
               #plcData.slots[#tempSlotNum].state := #STATE_FAULT;
           ELSIF (#statProblemPlcModulStates[#tempSlotNum + 1] = TRUE)
           THEN
               // Modul has a problem
               #plcData.slots[#tempSlotNum].faulty := FALSE;
               #plcData.slots[#tempSlotNum].problem := TRUE;
               #plcData.slots[#tempSlotNum].error := TRUE;
               #plcData.slots[#tempSlotNum].state := #STATE_PROBLEM;
           ELSE
               // Modul is OK
               #plcData.slots[#tempSlotNum].error := FALSE;
               #plcData.slots[#tempSlotNum].problem := FALSE;
               #plcData.slots[#tempSlotNum].faulty := FALSE;
           END_IF;

           // Error in PLC - Slot = 1, but index must be increased by 1, because of bit 0 = group display
           // --> used index = 2
           IF (#statProblemPlcModulStates[2] = TRUE)
               OR (#statFaultyPlcModulStates[2] = TRUE)
           THEN
               #plcData.error := TRUE;
           END_IF;
       END_IF;

       #tempSlotNum := #tempSlotNum + 1;
   END_WHILE;

   // Write static values to outputs
   #error := #statError;
   #status := #statStatus;
   #statusID := #statStatusID;

   //----------------------------------------------------------------------------------------------
END_FUNCTION_BLOCK

FUNCTION_BLOCK "NetDiag: IO Systems"   // FB30, SCL
{ S7_Optimized_Access := 'TRUE' }
VERSION : 0.1
   VAR_INPUT
      ioSystemHwId : Hw_IoSystem := 16#0000;   // This ID is representing the IO System (PN or DP), find the ID in the system constants
   END_VAR
   VAR_OUTPUT
      error : Bool := FALSE;   // Rising edge informs that an error occurred during the execution of the FB
      status : Word := 16#0000;   // Current status of FB
      statusID : Word := 16#0;   // Current status ID of calling instruction
   END_VAR
   VAR_IN_OUT
      ioSystemData : "UserDiag_typeIOSystem";   // IO-System diagnostics data
   END_VAR
   VAR
      statError : Bool := FALSE;   // Static value for output error
      statStatus : Word := 16#0000;   // Static value for output status
      statStatusID : Word := 16#0;   // Static value for output statusID
      statActualConfiguredDevices : Int := 0;   // Actual number of devices/slaves in the IOSystem/DP-Mastersystem
      statGeoAddr : GEOADDR;   // Slot information
      statGeoLaddr : Hw_Any := 16#0000;   // GEO2LOG hardware identifier
      statConfiguredDevices : Array[0..#DEVICES_STATES_UPPER_LIM] of Bool;   // Temporary storage of the return of "DeviceStates", to combine the states of the devices/slaves with numbers and names
      statExistingDevices : Array[0..#DEVICES_STATES_UPPER_LIM] of Bool;   // Temporary storage of the return of "DeviceStates", to combine the states of the devices/slaves with numbers and names
      statFaultyDevices : Array[0..#DEVICES_STATES_UPPER_LIM] of Bool;   // Temporary storage of the return of "DeviceStates", to combine the states of the devices/slaves with numbers and names
      statDisabledDevices : Array[0..#DEVICES_STATES_UPPER_LIM] of Bool;   // Temporary storage of the return of "DeviceStates", to combine the states of the devices/slaves with numbers and names
      statProblemDevices : Array[0..#DEVICES_STATES_UPPER_LIM] of Bool;   // Temporary storage of the return of "DeviceStates", to combine the states of the devices/slaves with numbers and names
      statDeviceProblemModules : Array[0..#MODULES_STATES_UPPER_LIM] of Bool;   // Storage of the status of all modules in the PN Devices / PB Slaves --> State: Problem
      statDeviceFaultyModules : Array[0..#MODULES_STATES_UPPER_LIM] of Bool;   // Storage of the status of all modules in the PN Devices / PB Slaves --> State: Faulty
      statDeviceExistingModules : Array[0..#MODULES_STATES_UPPER_LIM] of Bool;   // Storage of the status of all modules in the PN Devices / PB Slaves --> State: Existing
      instGetNameDevices : Get_Name;   // Instance of the system function "GetName"
      statInitString : String := '';   // Used to initialize the temporary string to convert into STRING[50]
      statFirstDevice : UInt := 0;   // Station number of the first device of the list
      statFirstDeviceFlag : Bool := TRUE;   // Help tag for the first device in the linked list
      statLastDevice : UInt := 0;   // Station number of the last device of the list
      statMaxDevices : Int := 0;   // Max devices per IO system
   END_VAR
   VAR_TEMP
      tempIndex : Int;   // Index of configured devices/slaves
      tempDeviceIndex : Int;   // Device/slave index
      tempSlotIndex : Int;   // Slot index
      tempSlotNum : Int;   // Index module number
      tempRetValGeo : Int;   // GEO2LOG error information
      tempRetValDeviceStates : Int;   // DeviceStates error information
      tempRetValModuleStates : Int;   // Return value of the system function "ModuleStates"
      tempStringConvert : String;   // Store the device names temporary here, to convert them into STRING[50]
      tempLastDevice : UInt;   // Temporary storage of the actual index, if it´s the last device --> store it in static
      tempDeviceInit : "UserDiag_typeDevice";   // Initalization of the device/slave diagnostic structure
   END_VAR
   VAR CONSTANT
      STATUS_EXECUTION_FINISHED : Word := 16#0000;   // Execution finished without errors
      ERR_MAX_SLOTS_PER_DEVICE : Word := 16#8400;   // There are more modules configured as defined with the user constant: USERDIAG_SLOTS_PER_DEVICE_UPPER_LIM
      ERR_MAX_DEVICES_PER_IOSYSTEM : Word := 16#8401;   // There are more modules configured as defined with the user constant: USERDIAG_DEVICES_PER_IO_SYTEM_UPPER_LIM
      ID_LOCAL : Word := 1;   // StatusID local
      ID_MODULE_STATES_CONFIGURED : Word := 2;   // StatusID during ModuleStates command (configured mode)
      ID_MODULE_STATES_FAULTY : Word := 3;   // StatusID during ModuleStates command (faulty mode)
      ID_MODULE_STATES_PROBLEM : Word := 4;   // StatusID during ModuleStates command (problem mode)
      ID_MODULE_STATES_EXISTING : Word := 5;   // StatusID during ModuleStates command (existing mode)
      ID_DEVICE_STATES_CONFIGURED : Word := 6;   // StatusID during DeviceStates command (configuration mode)
      ID_DEVICE_STATES_FAULTY : Word := 7;   // StatusID during DeviceStates command (fault mode)
      ID_DEVICE_STATES_PROBLEM : Word := 8;   // StatusID during DeviceStates command (problem mode)
      ID_DEVICE_STATES_EXISTING : Word := 9;   // StatusID during DeviceStates command (existing mode)
      ID_DEVICE_STATES_DISABLED : Word := 10;   // StatusID during DeviceStates command (disable mode)
      ID_GET_NAME : Word := 11;   // StatusID during GET_NAME command
      MODE_CONFIGURED : USInt := 1;   // Used for instruction DeviceStates/ModuleStates, read out all configured devices/slaves
      MODE_FAULTY : USInt := 2;   // Used for instruction DeviceStates/ModuleStates, read out all faulty devices/slaves
      MODE_DISABLED : USInt := 3;   // Used for instruction DeviceStates/ModuleStates, read out all disabled devices/slaves
      MODE_EXIST : USInt := 4;   // Used for instruction DeviceStates/ModuleStates, read out all devices/slaves not reachable
      MODE_PROBLEM : USInt := 5;   // Used for instruction DeviceStates/ModuleStates, read out all devices with several problems
      DEVICE_SLAVE : USInt := 2;   // GEO2LOG structure: HW type = 2
      MODULE_OF_DEVICE : USInt := 4;   // GEO2LOG structure: HW type = 4
      IO_SYSTEM_AREA : USInt := 1;   // GEO2LOG structure: Area = 1
      DP_SYSTEM_AREA : USInt := 2;   // GEO2LOG structure: Area = 2
      STATE_OK : USInt := 1;   // Device/modul state: ok
      STATE_FAULT : USInt := 2;   // Device/modul state: fault
      STATE_LOST_CON : USInt := 3;   // Device/modul state: lost connection
      STATE_DISABLED : USInt := 4;   // Device/modul state: disabled
      STATE_PROBLEM : USInt := 5;   // Device/modul state: problem
      STATE_WAS_FAULT : USInt := 12;   // Device/modul state: was fault
      STATE_WAS_LOST : USInt := 13;   // Device/modul state: connection was lost
      STATE_WAS_DISABLED : USInt := 14;   // Device/modul state: device/slave was disabled
      STATE_PROBLEM_GONE : USInt := 15;   // Device/modul state: had a problem
      MODULES_STATES_UPPER_LIM : Int := 127;   // Upper array limit for output tag of instruction ModuleStates
      DEVICES_STATES_UPPER_LIM : Int := 1023;   // Upper array limit for output tag of instruction DeviceStates
      ERR_HWID_NOT_EXISTENT : Int := 16#8091;   // Hardware identifier of the LADDR parameter does not exist. Check (for example, in the system constants) whether the value for LADDR exists in the project.
      ERR_LADDR_ADDRESS : Int := 16#8092;   // LADDR does not address a PROFINET IO or DP master system.
      POS_FIRST_CHAR : Int := 50;   // Position of first character to be deleted
      NUMBER_CHAR : Int := 204;   // Number of characters to be deleted
      MAX_SLAVES_DP : Int := 127;   // Max number of slaves in a PROFIBUS IO system
      LAST_DEVICE : Int := -1;   // No next device
   END_VAR
BEGIN
   //=============================================================================
   //SIEMENS AG
   //(c)Copyright 2015 All Rights Reserved
   //-----------------------------------------------------------------------------
   //Library: 
   //Tested with: S7-1516-3 PN/DP FW 2.5
   //Engineering: TIA Portal V15
   //Restrictions: Call in cyclic OB
   //Requirements: -
   //Functionality: Determine hardware identifier and module states from local and
   //               device modules 
   //-----------------------------------------------------------------------------
   //Change log table:
   //Version  Date       Expert in charge                Changes applied
   //01.00.00 27.01.2017 Siemens Industry Online Support First released version
   //01.00.01 20.12.2017 Siemens Industry Online Support GetStationInfo removed
   //01.00.02 27.02.2018 Siemens Industry Online Support Minor corrections
   //=============================================================================

   IF (#ioSystemHwId <> #ioSystemData.hardwareId)
   THEN
       // New IO System detected at input
       #statFirstDeviceFlag := TRUE;
       #statFirstDevice := 1;
       #statLastDevice := 1;

       #statActualConfiguredDevices := 0;
       #tempDeviceIndex := 1;

       #statError := FALSE;
       #statStatus := #STATUS_EXECUTION_FINISHED;
       #statStatusID := 0;
       #ioSystemData.error := FALSE;
       #ioSystemData.hardwareId := #ioSystemHwId;

       // Find out the number of the assigned IO system
       #tempRetValGeo := LOG2GEO(LADDR := #ioSystemHwId,
                                 GEOADDR := #statGeoAddr);
       // Set IO system ID
       #ioSystemData.number := #statGeoAddr.IOSYSTEM;

       // Initialize the structure for system function GEO2LOG
       #statGeoAddr.HWTYPE := #DEVICE_SLAVE;   // Hardware type 2: IO device

       // Predefine the type OF IO system. Either Profinet IO or Profibus DP
       IF (#statGeoAddr.AREA = #IO_SYSTEM_AREA)     // Area ID 1: PROFINET IO
       THEN
           #statMaxDevices := "USERDIAG_DEVICES_PER_IO_SYSTEM_UPPER_LIM";
       ELSIF (#statGeoAddr.AREA = #DP_SYSTEM_AREA) // Area ID 2: Profibus DP
       THEN
           IF ("USERDIAG_DEVICES_PER_IO_SYSTEM_UPPER_LIM" > #MAX_SLAVES_DP)
           THEN
               #statMaxDevices := #MAX_SLAVES_DP;
           ELSE
               #statMaxDevices := "USERDIAG_DEVICES_PER_IO_SYSTEM_UPPER_LIM";
           END_IF;
       ELSE
           #statMaxDevices := "USERDIAG_DEVICES_PER_IO_SYSTEM_UPPER_LIM";
       END_IF;

       // Set all other devices to not configured
       FOR #tempIndex := 1 TO "USERDIAG_DEVICES_PER_IO_SYSTEM_UPPER_LIM" DO
           #ioSystemData.devices[#tempIndex] := #tempDeviceInit;
       END_FOR;

       //=============================================================================
       // CONFIGURED DEVICES
       //=============================================================================
       // Find out how much devices are configured in the IO System --> PROFINET IO
       // This number is the maximum number of devices, which will be checked in the
       // following programm
       #tempRetValDeviceStates := DeviceStates(LADDR := #ioSystemHwId,
                                               MODE := #MODE_CONFIGURED,
                                               STATE := #statConfiguredDevices);

       // Check if the block call was successful
       IF (#tempRetValDeviceStates = 0)
       THEN
           // Call ok
           ;
       ELSIF (#tempRetValDeviceStates = #ERR_HWID_NOT_EXISTENT)
           OR (#tempRetValDeviceStates = #ERR_LADDR_ADDRESS)
       THEN
           #ioSystemData.error := TRUE;
           #statStatus := INT_TO_WORD(#tempRetValDeviceStates);
           #statStatusID := #ID_DEVICE_STATES_CONFIGURED;
           #statError := TRUE;
       ELSE
           // Error handling
           #statStatus := INT_TO_WORD(#tempRetValDeviceStates);
           #statStatusID := #ID_DEVICE_STATES_CONFIGURED;
           #statError := TRUE;
       END_IF;

       // Check if further devices are configured
       FOR #tempIndex := 1 TO #DEVICES_STATES_UPPER_LIM DO
           IF (((#statConfiguredDevices[#tempIndex] = TRUE)
               AND (#tempIndex > #statMaxDevices))
               AND (
               ((#statGeoAddr.AREA = #DP_SYSTEM_AREA)
               AND (#tempIndex < #MAX_SLAVES_DP))
               OR (#statGeoAddr.AREA = #IO_SYSTEM_AREA))
               )
           THEN
               // In the IOSystem are more devices configured as defined with the user constant
               #statStatus := #ERR_MAX_DEVICES_PER_IOSYSTEM;
               #statStatusID := #ID_LOCAL;
               #statError := TRUE;
           END_IF;
       END_FOR;

       //=============================================================================
       // Go trough all devices and get the status of the configured
       //=============================================================================
       FOR #tempIndex := 1 TO #statMaxDevices DO
           // The devices are configured --> Read out the logical address and the
           // device name
           IF (#statConfiguredDevices[#tempIndex] = TRUE)
           THEN
               // Store the first configured device for the linked list
               IF (#statFirstDeviceFlag = TRUE)
               THEN
                   #statFirstDevice := INT_TO_UINT(#tempIndex);
                   #ioSystemData.firstDevice := UINT_TO_INT(#statFirstDevice);
                   #statFirstDeviceFlag := FALSE;
                   #tempLastDevice := INT_TO_UINT(#tempIndex);
                   // It´s not the first bit --> Store the actual index as "next device"
                   // in the further one!
               ELSE
                   #ioSystemData.devices[#tempLastDevice].nextDevice := #tempIndex;
                   #tempLastDevice := INT_TO_UINT(#tempIndex);
               END_IF;
               // Store the index of the last device for the exit condition of the
               // followiing instructions
               #statLastDevice := #tempLastDevice;
               #ioSystemData.lastDevice := UINT_TO_INT(#statLastDevice);

               // Initialize the structure for system function GEO2LOG
               #statGeoAddr.STATION := INT_TO_UINT(#tempIndex); // Station number 
               #statGeoAddr.HWTYPE := #DEVICE_SLAVE;   // Hardware type 2: IO device

               // Read LADDR from devices
               #tempRetValGeo := GEO2LOG(GEOADDR := #statGeoAddr,
                                         LADDR => #statGeoLaddr);
               // Everything is ok!
               IF (#tempRetValGeo = 0)
               THEN
                   // Store LADDR from devices in diagnostics data block
                   #ioSystemData.devices[#tempIndex].hardwareId := #statGeoLaddr;
                   #ioSystemData.devices[#tempIndex].number := INT_TO_UINT(#tempIndex);
                   #ioSystemData.devices[#tempIndex].configured := TRUE;

                   // Store the device name, if the device is existing
                   // Get name is an acyclic instruction. In the startup OB, the
                   // instruction has to be repeated until it is done or error
                   REPEAT
                       // Get device name of each decive in PN System
                       #instGetNameDevices(LADDR := #ioSystemHwId,
                                           STATION_NR := #statGeoAddr.STATION,
                                           DATA := #tempStringConvert);

                   UNTIL ((#instGetNameDevices.DONE = TRUE)
                       OR (#instGetNameDevices.ERROR = TRUE))
                   END_REPEAT;

                   IF (#instGetNameDevices.ERROR = TRUE)
                   THEN
                       // Error handling
                       #statStatus := #instGetNameDevices.STATUS;
                       #statStatusID := #ID_GET_NAME;
                       #statError := TRUE;

                       // Everything is ok --> Convert the String[254] into String[50]    
                   ELSIF (#instGetNameDevices.DONE = TRUE)
                   THEN
                       // Cut all characters more than 50 to reduce the string length
                       #ioSystemData.devices[#tempIndex].name := STRING_TO_WSTRING(DELETE(IN := #tempStringConvert,
                                                                                          L := #NUMBER_CHAR,
                                                                                          P := #POS_FIRST_CHAR));

                       // Initialize the temporary string before next loop
                       #tempStringConvert := #statInitString;
                   ELSE
                       ;
                   END_IF;


                   //=============================================================================
                   // Get the logical address of all modules and store the actual number of
                   // modules from each device
                   //=============================================================================

                   // Initialize the structure for system function GEO2LOG
                   #statGeoAddr.HWTYPE := #MODULE_OF_DEVICE;   // Hardware type 4: Module

                   FOR #tempSlotNum := 0 TO "USERDIAG_SLOTS_PER_DEVICE_UPPER_LIM" DO
                       // Slot number
                       #statGeoAddr.SLOT := INT_TO_UINT(#tempSlotNum);
                       // read LADDR from modules
                       #tempRetValGeo := GEO2LOG(GEOADDR := #statGeoAddr,
                                                 LADDR => #statGeoLaddr);
                       // check Retval
                       IF (#tempRetValGeo = 0)
                       THEN
                           // Store LADDR from modules in diagnostic data block
                           #ioSystemData.devices[#tempIndex].slots[#tempSlotNum].hardwareId := #statGeoLaddr;
                           #ioSystemData.devices[#tempIndex].actualConfiguredSlots := #ioSystemData.devices[#tempIndex].actualConfiguredSlots + 1;

                           #ioSystemData.devices[#tempIndex].slots[#tempSlotNum].configured := TRUE;

                       ELSE
                           // If the return value is not 0 --> the device/system/module is
                           // not configured --> No error handling
                           // set LADDR from modules to 0 in diagnostic data block
                           #ioSystemData.devices[#tempIndex].slots[#tempSlotNum].hardwareId := 0;
                       END_IF;
                   END_FOR;

                   // Check if further slots are configured
                   #statGeoAddr.SLOT := INT_TO_UINT(#tempSlotNum);

                   #tempRetValGeo := GEO2LOG(GEOADDR := #statGeoAddr,
                                             LADDR => #statGeoLaddr);

                   IF ((#tempRetValGeo = 0)
                       AND (#statGeoLaddr <> 16#0))
                   THEN
                       // In the PLC are more slots configured as defined with the user constant
                       #statStatus := #ERR_MAX_SLOTS_PER_DEVICE;
                       #statStatusID := #ID_LOCAL;
                       #statError := TRUE;
                   END_IF;

                   // Increment the actual configured devices, store the state and
                   // HW_ID as an numerical value (UINT)
                   #statActualConfiguredDevices := #statActualConfiguredDevices + 1;
               ELSE
                   ;
               END_IF;

           ELSE
               ; // Device not configured
           END_IF;
       END_FOR;

       #ioSystemData.actualConfiguredDevices := #statActualConfiguredDevices;

       // Mark parameter "Next Device" of the last device in the list
       // --> "Next Device" = negative --> Last device in the list
       #ioSystemData.devices[#statLastDevice].nextDevice := #LAST_DEVICE;

   END_IF; // New IO System detected at input

   #ioSystemData.error := FALSE; // Reset the IO-System error status


   //=============================================================================
   // START DIAGNOSTICS EVALUATION
   //=============================================================================

   //=============================================================================
   // EXISTING DEVICES
   //=============================================================================
   #tempRetValDeviceStates := DeviceStates(LADDR := #ioSystemHwId,
                                           MODE := #MODE_EXIST,
                                           STATE := #statExistingDevices);

   // Check if the block call was successful
   IF (#tempRetValDeviceStates = 0)
   THEN
       // Call ok 
       ;
   ELSIF ((#tempRetValDeviceStates = #ERR_HWID_NOT_EXISTENT)
       OR (#tempRetValDeviceStates = #ERR_LADDR_ADDRESS))
   THEN
       #ioSystemData.error := TRUE;
       #statStatus := INT_TO_WORD(#tempRetValDeviceStates);
       #statStatusID := #ID_DEVICE_STATES_EXISTING;
       #statError := TRUE;
   ELSE
       // Error handling
       #statStatus := INT_TO_WORD(#tempRetValDeviceStates);
       #statStatusID := #ID_DEVICE_STATES_EXISTING;
       #statError := TRUE;
   END_IF;

   //=============================================================================
   // FAULTY DEVICES
   //=============================================================================
   #tempRetValDeviceStates := DeviceStates(LADDR := #ioSystemHwId,
                                           MODE := #MODE_FAULTY,
                                           STATE := #statFaultyDevices);

   // Check if the block call was successful
   IF (#tempRetValDeviceStates = 0)
   THEN
       // Call ok
       ;
   ELSIF ((#tempRetValDeviceStates = #ERR_HWID_NOT_EXISTENT)
       OR (#tempRetValDeviceStates = #ERR_LADDR_ADDRESS))
   THEN
       #ioSystemData.error := TRUE;
       #statStatus := INT_TO_WORD(#tempRetValDeviceStates);
       #statStatusID := #ID_DEVICE_STATES_FAULTY;
       #statError := TRUE;
   ELSE
       // Error handling
       #statStatus := INT_TO_WORD(#tempRetValDeviceStates);
       #statStatusID := #ID_DEVICE_STATES_FAULTY;
       #statError := TRUE;
   END_IF;

   //=============================================================================
   // DISABLED DEVICES
   //=============================================================================
   #tempRetValDeviceStates := DeviceStates(LADDR := #ioSystemHwId,
                                           MODE := #MODE_DISABLED,
                                           STATE := #statDisabledDevices);

   // Check if the block call was successful
   IF (#tempRetValDeviceStates = 0)
   THEN
       // Call ok
       ;
   ELSIF ((#tempRetValDeviceStates = #ERR_HWID_NOT_EXISTENT)
       OR (#tempRetValDeviceStates = #ERR_LADDR_ADDRESS))
   THEN
       #ioSystemData.error := TRUE;
       #statStatus := INT_TO_WORD(#tempRetValDeviceStates);
       #statStatusID := #ID_DEVICE_STATES_DISABLED;
       #statError := TRUE;
   ELSE
       // Error handling
       #statStatus := INT_TO_WORD(#tempRetValDeviceStates);
       #statStatusID := #ID_DEVICE_STATES_DISABLED;
       #statError := TRUE;
   END_IF;

   //=============================================================================
   // PROBLEM DEVICES
   //=============================================================================
   #tempRetValDeviceStates := DeviceStates(LADDR := #ioSystemHwId,
                                           MODE := #MODE_PROBLEM,
                                           STATE := #statProblemDevices);

   // Check if the block call was successful
   IF (#tempRetValDeviceStates = 0)
   THEN
       // Call ok
       ;
   ELSIF ((#tempRetValDeviceStates = #ERR_HWID_NOT_EXISTENT)
       OR (#tempRetValDeviceStates = #ERR_LADDR_ADDRESS))
   THEN
       #ioSystemData.error := TRUE;
       #statStatus := INT_TO_WORD(#tempRetValDeviceStates);
       #statStatusID := #ID_DEVICE_STATES_PROBLEM;
       #statError := TRUE;
   ELSE
       // Error handling
       #statStatus := INT_TO_WORD(#tempRetValDeviceStates);
       #statStatusID := #ID_DEVICE_STATES_PROBLEM;
       #statError := TRUE;
   END_IF;

   //=============================================================================
   // Go through configured devices and check for error
   //=============================================================================
   // Initialize the pointer for the first run 
   #tempDeviceIndex := #ioSystemData.firstDevice;

   WHILE ((#tempDeviceIndex <= "USERDIAG_DEVICES_PER_IO_SYSTEM_UPPER_LIM")
       AND (#tempDeviceIndex > 0))
   DO

       IF (#ioSystemData.devices[#tempDeviceIndex].configured = TRUE)
       THEN

           IF (#statDisabledDevices[#tempDeviceIndex] = TRUE)
           THEN
               //===================
               // Device is disabled
               //===================
               #ioSystemData.devices[#tempDeviceIndex].disabled := TRUE;
               #ioSystemData.devices[#tempDeviceIndex].error := FALSE;
               #ioSystemData.devices[#tempDeviceIndex].faulty := FALSE;
               #ioSystemData.devices[#tempDeviceIndex].problem := FALSE;
               #ioSystemData.devices[#tempDeviceIndex].state := #STATE_DISABLED;

           ELSE
               #ioSystemData.devices[#tempDeviceIndex].disabled := FALSE;

               IF (#statExistingDevices[#tempDeviceIndex] = TRUE)
               THEN
                   #ioSystemData.devices[#tempDeviceIndex].exists := TRUE;

                   CASE #ioSystemData.devices[#tempDeviceIndex].state OF
                       #STATE_WAS_FAULT,
                       #STATE_WAS_LOST,
                       #STATE_WAS_DISABLED,
                       #STATE_PROBLEM_GONE:
                           ;
                       #STATE_FAULT:
                           #ioSystemData.devices[#tempDeviceIndex].state := #STATE_WAS_FAULT;
                       #STATE_LOST_CON:
                           #ioSystemData.devices[#tempDeviceIndex].state := #STATE_WAS_LOST;
                       #STATE_DISABLED:
                           #ioSystemData.devices[#tempDeviceIndex].state := #STATE_WAS_DISABLED;
                       #STATE_PROBLEM:
                           #ioSystemData.devices[#tempDeviceIndex].state := #STATE_PROBLEM_GONE;
                       ELSE
                           #ioSystemData.devices[#tempDeviceIndex].state := #STATE_OK;
                   END_CASE;

               ELSE
                   // Device not existent
                   #ioSystemData.devices[#tempDeviceIndex].error := TRUE;
                   #ioSystemData.error := TRUE;
                   #ioSystemData.devices[#tempDeviceIndex].exists := FALSE;
               END_IF; // End: Device exists


               IF (#statFaultyDevices[#tempDeviceIndex] = FALSE)
               THEN
                   // Device is not faulty
                   #ioSystemData.devices[#tempDeviceIndex].error := FALSE;
                   #ioSystemData.devices[#tempDeviceIndex].faulty := FALSE;

                   IF (#statProblemDevices[#tempDeviceIndex] = FALSE)
                   THEN
                       //============================
                       // Device has no problem
                       //============================
                       #ioSystemData.devices[#tempDeviceIndex].error := FALSE;
                       #ioSystemData.devices[#tempDeviceIndex].problem := FALSE;
                   ELSE
                       //============================
                       // Device has a problem
                       //============================
                       #ioSystemData.devices[#tempDeviceIndex].error := TRUE;
                       #ioSystemData.error := TRUE;
                       #ioSystemData.devices[#tempDeviceIndex].problem := TRUE;
                       #ioSystemData.devices[#tempDeviceIndex].state := #STATE_PROBLEM;
                   END_IF;

               ELSE
                   // Device is faulty, don't matter what happened
                   #ioSystemData.devices[#tempDeviceIndex].error := TRUE;
                   #ioSystemData.error := TRUE;
                   #ioSystemData.devices[#tempDeviceIndex].faulty := TRUE;

                   IF (#statProblemDevices[#tempDeviceIndex] = FALSE)
                   THEN
                       //============================
                       // Device has no problem
                       //============================
                       #ioSystemData.devices[#tempDeviceIndex].problem := FALSE;
                   ELSE
                       //============================
                       // Device has a problem
                       //============================
                       #ioSystemData.devices[#tempDeviceIndex].problem := TRUE;
                   END_IF;

                   IF (#statExistingDevices[#tempDeviceIndex] = FALSE)
                   THEN
                       //==========================
                       // Device is lost
                       //==========================
                       #ioSystemData.devices[#tempDeviceIndex].state := #STATE_LOST_CON;
                       #ioSystemData.devices[#tempDeviceIndex].exists := FALSE;
                   ELSE
                       //==========================
                       // Device is faulty
                       //==========================
                       #ioSystemData.devices[#tempDeviceIndex].state := #STATE_FAULT;
                       #ioSystemData.devices[#tempDeviceIndex].exists := TRUE;
                   END_IF;
               END_IF; // End: // Device is not faulty

           END_IF;

           //=============================================================================
           // Set module states
           //=============================================================================
           // Check ModuleStates if device has a problem or is faulty
           IF ((#ioSystemData.devices[#tempDeviceIndex].problem = TRUE)
               OR (#ioSystemData.devices[#tempDeviceIndex].faulty = TRUE))
           THEN

               // PROBLEM MODULE
               #tempRetValModuleStates := ModuleStates(LADDR := #ioSystemData.devices[#tempDeviceIndex].hardwareId,
                                                       MODE := #MODE_PROBLEM,
                                                       STATE := #statDeviceProblemModules);

               // Check if the block call was successful
               IF (#tempRetValModuleStates = 0)
               THEN
                   // Call ok 
                   ;
               ELSIF ((#tempRetValModuleStates = #ERR_HWID_NOT_EXISTENT)
                   OR (#tempRetValModuleStates = #ERR_LADDR_ADDRESS))
               THEN
                   #ioSystemData.error := TRUE;
                   #statStatus := INT_TO_WORD(#tempRetValModuleStates);
                   #statStatusID := #ID_MODULE_STATES_PROBLEM;
                   #statError := TRUE;
               ELSE
                   // Error handling
                   #statStatus := INT_TO_WORD(#tempRetValModuleStates);
                   #statStatusID := #ID_MODULE_STATES_PROBLEM;
                   #statError := TRUE;
               END_IF;

               // FAULTY MODULE
               #tempRetValModuleStates := ModuleStates(LADDR := #ioSystemData.devices[#tempDeviceIndex].hardwareId,
                                                       MODE := #MODE_FAULTY,
                                                       STATE := #statDeviceFaultyModules);

               // Check if the block call was successful
               IF (#tempRetValModuleStates = 0)
               THEN
                   // Call ok 
                   ;
               ELSIF ((#tempRetValModuleStates = #ERR_HWID_NOT_EXISTENT)
                   OR (#tempRetValModuleStates = #ERR_LADDR_ADDRESS))
               THEN
                   #ioSystemData.error := TRUE;
                   #statStatus := INT_TO_WORD(#tempRetValModuleStates);
                   #statStatusID := #ID_MODULE_STATES_FAULTY;
                   #statError := TRUE;
               ELSE
                   // Error handling
                   #statStatus := INT_TO_WORD(#tempRetValModuleStates);
                   #statStatusID := #ID_MODULE_STATES_FAULTY;
                   #statError := TRUE;
               END_IF;

               // EXISTING MODULE
               #tempRetValModuleStates := ModuleStates(LADDR := #ioSystemData.devices[#tempDeviceIndex].hardwareId,
                                                       MODE := #MODE_EXIST,
                                                       STATE := #statDeviceExistingModules);

               // Check if the block call was successful
               IF (#tempRetValModuleStates = 0)
               THEN
                   // Call ok 
                   ;
               ELSIF ((#tempRetValModuleStates = #ERR_HWID_NOT_EXISTENT)
                   OR (#tempRetValModuleStates = #ERR_LADDR_ADDRESS))
               THEN
                   #ioSystemData.error := TRUE;
                   #statStatus := INT_TO_WORD(#tempRetValModuleStates);
                   #statStatusID := #ID_MODULE_STATES_EXISTING;
                   #statError := TRUE;
               ELSE
                   // Error handling
                   #statStatus := INT_TO_WORD(#tempRetValModuleStates);
                   #statStatusID := #ID_MODULE_STATES_EXISTING;
                   #statError := TRUE;
               END_IF;
           END_IF;


           FOR #tempSlotIndex := 0 TO "USERDIAG_SLOTS_PER_DEVICE_UPPER_LIM" DO
               IF (#ioSystemData.devices[#tempDeviceIndex].slots[#tempSlotIndex].configured = TRUE)
               THEN
                   CASE #ioSystemData.devices[#tempDeviceIndex].slots[#tempSlotIndex].state OF
                       #STATE_WAS_FAULT,
                       #STATE_WAS_LOST,
                       #STATE_WAS_DISABLED,
                       #STATE_PROBLEM_GONE:
                           ;
                       #STATE_FAULT:
                           #ioSystemData.devices[#tempDeviceIndex].slots[#tempSlotIndex].state := #STATE_WAS_FAULT;
                       #STATE_LOST_CON:
                           #ioSystemData.devices[#tempDeviceIndex].slots[#tempSlotIndex].state := #STATE_WAS_LOST;
                       #STATE_DISABLED:
                           #ioSystemData.devices[#tempDeviceIndex].slots[#tempSlotIndex].state := #STATE_WAS_DISABLED;
                       #STATE_PROBLEM:
                           #ioSystemData.devices[#tempDeviceIndex].slots[#tempSlotIndex].state := #STATE_PROBLEM_GONE;
                       ELSE
                           #ioSystemData.devices[#tempDeviceIndex].slots[#tempSlotIndex].state := #STATE_OK;
                   END_CASE;
               END_IF;
           END_FOR;

           CASE #ioSystemData.devices[#tempDeviceIndex].state OF

               #STATE_DISABLED:
                   FOR #tempSlotIndex := 0 TO "USERDIAG_SLOTS_PER_DEVICE_UPPER_LIM" DO
                       IF (#ioSystemData.devices[#tempDeviceIndex].slots[#tempSlotIndex].configured = TRUE)
                       THEN
                           //NEW: Set all configured modules of device to disabled
                           #ioSystemData.devices[#tempDeviceIndex].slots[#tempSlotIndex].disabled := TRUE;
                           #ioSystemData.devices[#tempDeviceIndex].slots[#tempSlotIndex].error := FALSE;
                           #ioSystemData.devices[#tempDeviceIndex].slots[#tempSlotIndex].faulty := FALSE;
                           #ioSystemData.devices[#tempDeviceIndex].slots[#tempSlotIndex].problem := FALSE;
                           #ioSystemData.devices[#tempDeviceIndex].slots[#tempSlotIndex].state := #STATE_DISABLED;
                       END_IF;
                   END_FOR;

               #STATE_LOST_CON:
                   // All modules are faulty when connection is lost
                   FOR #tempSlotIndex := 0 TO "USERDIAG_SLOTS_PER_DEVICE_UPPER_LIM" DO
                       IF (#ioSystemData.devices[#tempDeviceIndex].slots[#tempSlotIndex].configured = TRUE)
                       THEN
                           #ioSystemData.devices[#tempDeviceIndex].slots[#tempSlotIndex].error := TRUE;
                           #ioSystemData.devices[#tempDeviceIndex].slots[#tempSlotIndex].faulty := TRUE;
                           #ioSystemData.devices[#tempDeviceIndex].slots[#tempSlotIndex].problem := TRUE;
                           #ioSystemData.devices[#tempDeviceIndex].slots[#tempSlotIndex].exists := FALSE;
                           #ioSystemData.devices[#tempDeviceIndex].slots[#tempSlotIndex].state := #STATE_LOST_CON;
                       END_IF;
                   END_FOR;

               #STATE_FAULT,
               #STATE_PROBLEM:
                   // The device is reachable, but faulty because of an error in a
                   // subordinated system --> check the modules
                   // Store the state of the different module in the diag DB
                   FOR #tempSlotIndex := 0 TO "USERDIAG_SLOTS_PER_DEVICE_UPPER_LIM" DO
                       IF (#ioSystemData.devices[#tempDeviceIndex].slots[#tempSlotIndex].configured = TRUE)
                       THEN
                           IF (#statDeviceProblemModules[#tempSlotIndex + 1] = TRUE)
                           THEN
                               // Problem in module
                               #ioSystemData.devices[#tempDeviceIndex].slots[#tempSlotIndex].faulty := FALSE;
                               #ioSystemData.devices[#tempDeviceIndex].slots[#tempSlotIndex].error := TRUE;
                               #ioSystemData.devices[#tempDeviceIndex].slots[#tempSlotIndex].problem := TRUE;
                               #ioSystemData.devices[#tempDeviceIndex].slots[#tempSlotIndex].state := #STATE_PROBLEM;

